// TIA Portal V15.1 export
// export: Created 2024-05-17T05:38:55.5837031Z, ExportSetting WithDefaults, DisplayName Totally Integrated Automation Portal, DisplayVersion V15.1 Update 5, DisplayName TIA Portal Openness, DisplayVersion V15.1 Update 5, DisplayName SINAMICS Startdrive Advanced, DisplayVersion V15.1, DisplayName G130, G150, S120, S150, SINAMICS MV, S210, DisplayVersion V15.1, DisplayName G110M, G120, G120C, G120D, G120P, DisplayVersion V15.1, DisplayName STEP 7 Professional, DisplayVersion V15.1 Update 5, DisplayName STEP 7 Safety, DisplayVersion V15.1, DisplayName WinCC Professional, DisplayVersion V15.1 Update 5, DisplayName SIMATIC Visualization Architect, DisplayVersion V15.1
FUNCTION "209220ZM01DataHandling" : Void   // FC354, FBD
TITLE = 209220ZM01 Data Handling
{ S7_Optimized_Access := 'FALSE' }
AUTHOR : VCC
VERSION : 0.1
// stored: AutoNumber false, IsIECCheckEnabled false, SetENOAutomatically False, UDAEnableTagReadback false
   VAR_OUTPUT
      O_AlarmA : Bool;   // Alarm A
      O_AlarmB : Bool;   // Alarm B
      O_AlarmC : Bool;   // Alarm C
      O_AlarmD : Bool;   // Alarm D
      O_AlarmABCondition : Bool;   // Alarm AB Condition
      H_IAnim : Word;   // Icon Animation
   END_VAR
BEGIN

REGION Network 1: **** 4.6 - Machine status - Indications **** Icon animation
   // Icon animation
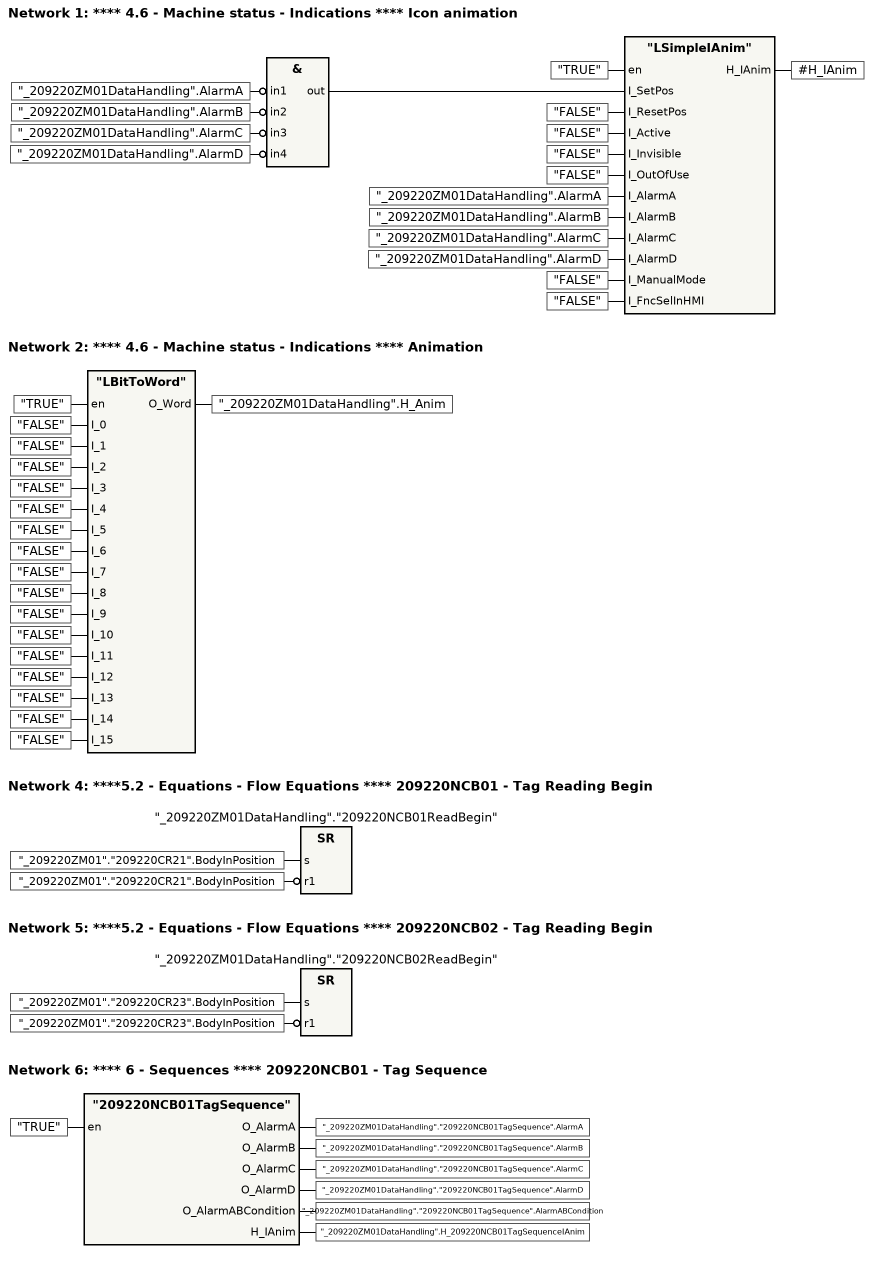
   IF "TRUE" THEN
       "LSimpleIAnim"(I_SetPos := NOT "_209220ZM01DataHandling".AlarmA AND NOT "_209220ZM01DataHandling".AlarmB AND NOT "_209220ZM01DataHandling".AlarmC AND NOT "_209220ZM01DataHandling".AlarmD,
                      I_ResetPos := "FALSE",
                      I_Active := "FALSE",
                      I_Invisible := "FALSE",
                      I_OutOfUse := "FALSE",
                      I_AlarmA := "_209220ZM01DataHandling".AlarmA,
                      I_AlarmB := "_209220ZM01DataHandling".AlarmB,
                      I_AlarmC := "_209220ZM01DataHandling".AlarmC,
                      I_AlarmD := "_209220ZM01DataHandling".AlarmD,
                      I_ManualMode := "FALSE",
                      I_FncSelInHMI := "FALSE",
                      H_IAnim => #H_IAnim);
   END_IF;
END_REGION

REGION Network 2: **** 4.6 - Machine status - Indications **** Animation
   // Animation
   IF "TRUE" THEN
       "LBitToWord"(I_0 := "FALSE",
                    I_1 := "FALSE",
                    I_2 := "FALSE",
                    I_3 := "FALSE",
                    I_4 := "FALSE",
                    I_5 := "FALSE",
                    I_6 := "FALSE",
                    I_7 := "FALSE",
                    I_8 := "FALSE",
                    I_9 := "FALSE",
                    I_10 := "FALSE",
                    I_11 := "FALSE",
                    I_12 := "FALSE",
                    I_13 := "FALSE",
                    I_14 := "FALSE",
                    I_15 := "FALSE",
                    O_Word => "_209220ZM01DataHandling".H_Anim);
   END_IF;
END_REGION

NETWORK
TITLE = **** 4.6 - Machine Status - Indications **** Animation DB number
// DB number
      OPN   "_209220ZM01DataHandling";
      L     DBNO;
      T     "_209220ZM01DataHandling".H_DBnr;

REGION Network 4: ****5.2 - Equations - Flow Equations **** 209220NCB01 - Tag Reading Begin
   // Singal to start the reading of the Tag
   IF "_209220ZM01"."209220CR21".BodyInPosition THEN
       "_209220ZM01DataHandling"."209220NCB01ReadBegin" := TRUE;   // SR flip-flop
   END_IF;
   IF NOT "_209220ZM01"."209220CR21".BodyInPosition THEN
       "_209220ZM01DataHandling"."209220NCB01ReadBegin" := FALSE;
   END_IF;
END_REGION

REGION Network 5: ****5.2 - Equations - Flow Equations **** 209220NCB02 - Tag Reading Begin
   // Singal to start the reading of the Tag
   IF "_209220ZM01"."209220CR23".BodyInPosition THEN
       "_209220ZM01DataHandling"."209220NCB02ReadBegin" := TRUE;   // SR flip-flop
   END_IF;
   IF NOT "_209220ZM01"."209220CR23".BodyInPosition THEN
       "_209220ZM01DataHandling"."209220NCB02ReadBegin" := FALSE;
   END_IF;
END_REGION

REGION Network 6: **** 6 - Sequences **** 209220NCB01 - Tag Sequence
   // Tag Sequence
   IF "TRUE" THEN
       "209220NCB01TagSequence"(O_AlarmA => "_209220ZM01DataHandling"."209220NCB01TagSequence".AlarmA,
                               O_AlarmB => "_209220ZM01DataHandling"."209220NCB01TagSequence".AlarmB,
                               O_AlarmC => "_209220ZM01DataHandling"."209220NCB01TagSequence".AlarmC,
                               O_AlarmD => "_209220ZM01DataHandling"."209220NCB01TagSequence".AlarmD,
                               O_AlarmABCondition => "_209220ZM01DataHandling"."209220NCB01TagSequence".AlarmABCondition,
                               H_IAnim => "_209220ZM01DataHandling".H_209220NCB01TagSequenceIAnim);
   END_IF;
END_REGION

REGION Network 7: **** 6 - Sequences **** 209220NCB02 - Tag Sequence
   // Tag Sequence
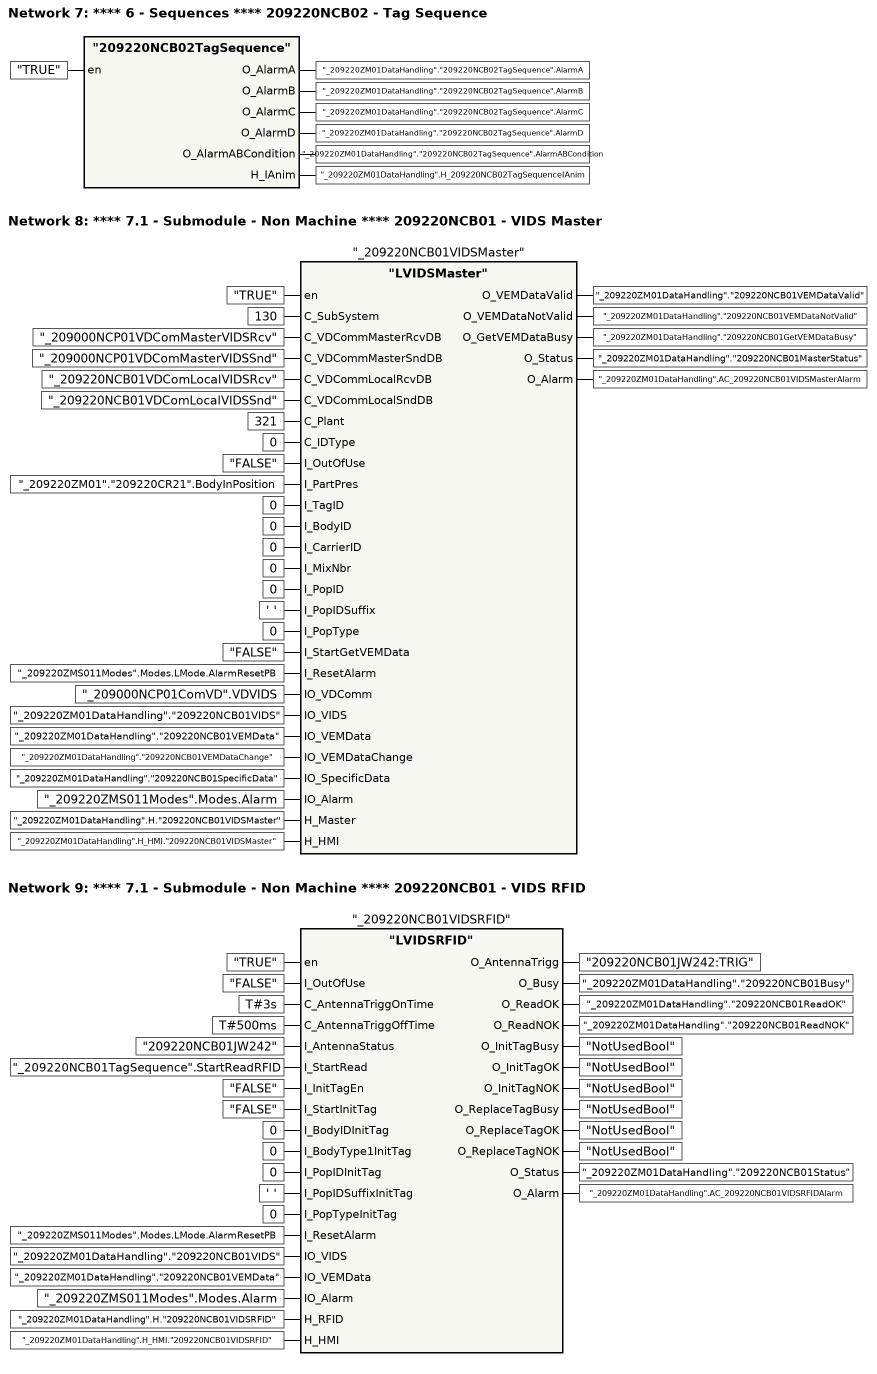
   IF "TRUE" THEN
       "209220NCB02TagSequence"(O_AlarmA => "_209220ZM01DataHandling"."209220NCB02TagSequence".AlarmA,
                               O_AlarmB => "_209220ZM01DataHandling"."209220NCB02TagSequence".AlarmB,
                               O_AlarmC => "_209220ZM01DataHandling"."209220NCB02TagSequence".AlarmC,
                               O_AlarmD => "_209220ZM01DataHandling"."209220NCB02TagSequence".AlarmD,
                               O_AlarmABCondition => "_209220ZM01DataHandling"."209220NCB02TagSequence".AlarmABCondition,
                               H_IAnim => "_209220ZM01DataHandling".H_209220NCB02TagSequenceIAnim);
   END_IF;
END_REGION

REGION Network 8: **** 7.1 - Submodule - Non Machine **** 209220NCB01 - VIDS Master
   // VIDS Master Module
   IF "TRUE" THEN
       "_209220NCB01VIDSMaster"(C_SubSystem := 130,   // "LVIDSMaster"
                               C_VDCommMasterRcvDB := "_209000NCP01VDComMasterVIDSRcv",
                               C_VDCommMasterSndDB := "_209000NCP01VDComMasterVIDSSnd",
                               C_VDCommLocalRcvDB := "_209220NCB01VDComLocalVIDSRcv",
                               C_VDCommLocalSndDB := "_209220NCB01VDComLocalVIDSSnd",
                               C_Plant := 321,
                               C_IDType := 0,
                               I_OutOfUse := "FALSE",
                               I_PartPres := "_209220ZM01"."209220CR21".BodyInPosition,
                               I_TagID := 0,
                               I_BodyID := 0,
                               I_CarrierID := 0,
                               I_MixNbr := 0,
                               I_PopID := 0,
                               I_PopIDSuffix := ' ',
                               I_PopType := 0,
                               I_StartGetVEMData := "FALSE",
                               I_ResetAlarm := "_209220ZMS011Modes".Modes.LMode.AlarmResetPB,
                               IO_VDComm := "_209000NCP01ComVD".VDVIDS,
                               IO_VIDS := "_209220ZM01DataHandling"."209220NCB01VIDS",
                               IO_VEMData := "_209220ZM01DataHandling"."209220NCB01VEMData",
                               IO_VEMDataChange := "_209220ZM01DataHandling"."209220NCB01VEMDataChange",
                               IO_SpecificData := "_209220ZM01DataHandling"."209220NCB01SpecificData",
                               IO_Alarm := "_209220ZMS011Modes".Modes.Alarm,
                               H_Master := "_209220ZM01DataHandling".H."209220NCB01VIDSMaster",
                               H_HMI := "_209220ZM01DataHandling".H_HMI."209220NCB01VIDSMaster",
                               O_VEMDataValid => "_209220ZM01DataHandling"."209220NCB01VEMDataValid",
                               O_VEMDataNotValid => "_209220ZM01DataHandling"."209220NCB01VEMDataNotValid",
                               O_GetVEMDataBusy => "_209220ZM01DataHandling"."209220NCB01GetVEMDataBusy",
                               O_Status => "_209220ZM01DataHandling"."209220NCB01MasterStatus",
                               O_Alarm => "_209220ZM01DataHandling".AC_209220NCB01VIDSMasterAlarm);
   END_IF;
END_REGION

REGION Network 9: **** 7.1 - Submodule - Non Machine **** 209220NCB01 - VIDS RFID
   // VIDS RFID Module
   IF "TRUE" THEN
       "_209220NCB01VIDSRFID"(I_OutOfUse := "FALSE",   // "LVIDSRFID"
                              C_AntennaTriggOnTime := T#3s,
                              C_AntennaTriggOffTime := T#500ms,
                              I_AntennaStatus := "209220NCB01JW242",
                              I_StartRead := "_209220NCB01TagSequence".StartReadRFID,
                              I_InitTagEn := "FALSE",
                              I_StartInitTag := "FALSE",
                              I_BodyIDInitTag := 0,
                              I_BodyType1InitTag := 0,
                              I_PopIDInitTag := 0,
                              I_PopIDSuffixInitTag := ' ',
                              I_PopTypeInitTag := 0,
                              I_ResetAlarm := "_209220ZMS011Modes".Modes.LMode.AlarmResetPB,
                              IO_VIDS := "_209220ZM01DataHandling"."209220NCB01VIDS",
                              IO_VEMData := "_209220ZM01DataHandling"."209220NCB01VEMData",
                              IO_Alarm := "_209220ZMS011Modes".Modes.Alarm,
                              H_RFID := "_209220ZM01DataHandling".H."209220NCB01VIDSRFID",
                              H_HMI := "_209220ZM01DataHandling".H_HMI."209220NCB01VIDSRFID",
                              O_AntennaTrigg => "209220NCB01JW242:TRIG",
                              O_Busy => "_209220ZM01DataHandling"."209220NCB01Busy",
                              O_ReadOK => "_209220ZM01DataHandling"."209220NCB01ReadOK",
                              O_ReadNOK => "_209220ZM01DataHandling"."209220NCB01ReadNOK",
                              O_InitTagBusy => "NotUsedBool",
                              O_InitTagOK => "NotUsedBool",
                              O_InitTagNOK => "NotUsedBool",
                              O_ReplaceTagBusy => "NotUsedBool",
                              O_ReplaceTagOK => "NotUsedBool",
                              O_ReplaceTagNOK => "NotUsedBool",
                              O_Status => "_209220ZM01DataHandling"."209220NCB01Status",
                              O_Alarm => "_209220ZM01DataHandling".AC_209220NCB01VIDSRFIDAlarm);
   END_IF;
END_REGION

REGION Network 10: **** 7.1 - Submodule - Non Machine ****209220NCB01 - VIDS Tracking
   // VIDS Tracking Module
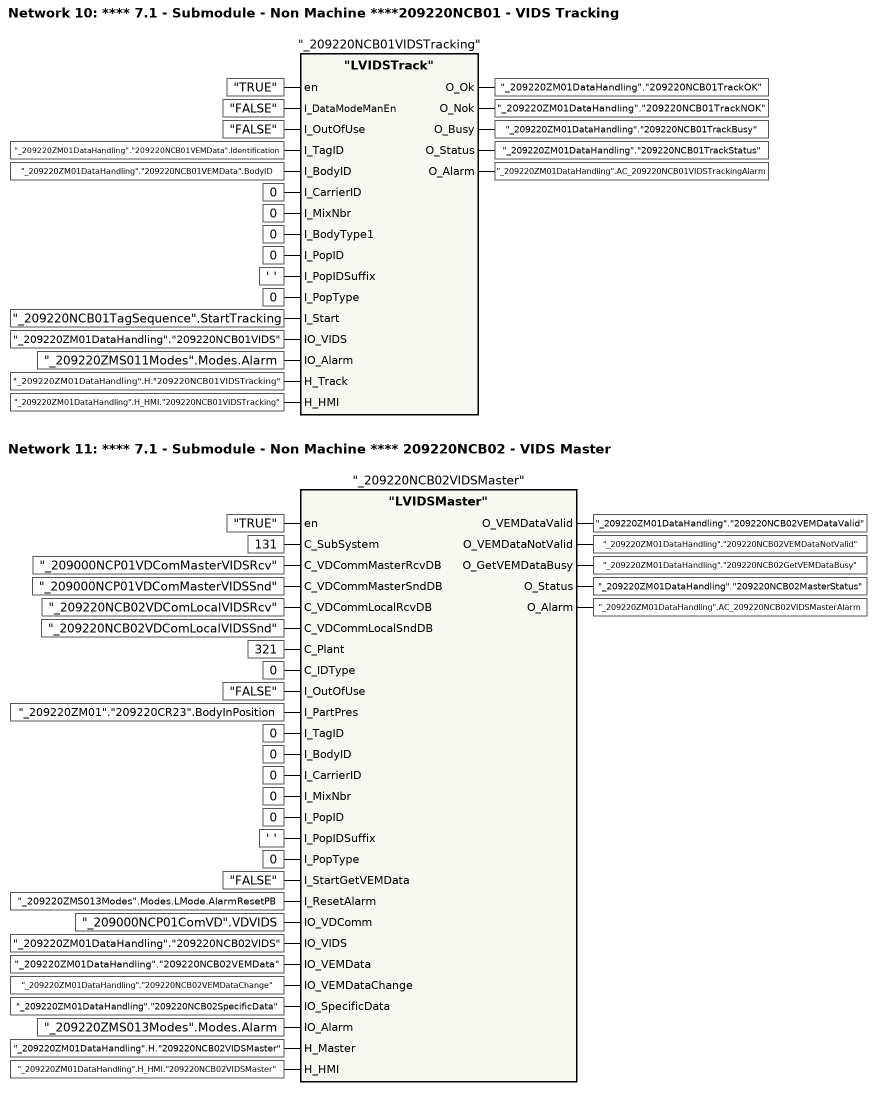
   IF "TRUE" THEN
       "_209220NCB01VIDSTracking"(I_DataModeManEn := "FALSE",   // "LVIDSTrack"
                               I_OutOfUse := "FALSE",
                               I_TagID := "_209220ZM01DataHandling"."209220NCB01VEMData".Identification,
                               I_BodyID := "_209220ZM01DataHandling"."209220NCB01VEMData".BodyID,
                               I_CarrierID := 0,
                               I_MixNbr := 0,
                               I_BodyType1 := 0,
                               I_PopID := 0,
                               I_PopIDSuffix := ' ',
                               I_PopType := 0,
                               I_Start := "_209220NCB01TagSequence".StartTracking,
                               IO_VIDS := "_209220ZM01DataHandling"."209220NCB01VIDS",
                               IO_Alarm := "_209220ZMS011Modes".Modes.Alarm,
                               H_Track := "_209220ZM01DataHandling".H."209220NCB01VIDSTracking",
                               H_HMI := "_209220ZM01DataHandling".H_HMI."209220NCB01VIDSTracking",
                               O_Ok => "_209220ZM01DataHandling"."209220NCB01TrackOK",
                               O_Nok => "_209220ZM01DataHandling"."209220NCB01TrackNOK",
                               O_Busy => "_209220ZM01DataHandling"."209220NCB01TrackBusy",
                               O_Status => "_209220ZM01DataHandling"."209220NCB01TrackStatus",
                               O_Alarm => "_209220ZM01DataHandling".AC_209220NCB01VIDSTrackingAlarm);
   END_IF;
END_REGION

REGION Network 11: **** 7.1 - Submodule - Non Machine **** 209220NCB02 - VIDS Master
   // VIDS Master Module
   IF "TRUE" THEN
       "_209220NCB02VIDSMaster"(C_SubSystem := 131,   // "LVIDSMaster"
                               C_VDCommMasterRcvDB := "_209000NCP01VDComMasterVIDSRcv",
                               C_VDCommMasterSndDB := "_209000NCP01VDComMasterVIDSSnd",
                               C_VDCommLocalRcvDB := "_209220NCB02VDComLocalVIDSRcv",
                               C_VDCommLocalSndDB := "_209220NCB02VDComLocalVIDSSnd",
                               C_Plant := 321,
                               C_IDType := 0,
                               I_OutOfUse := "FALSE",
                               I_PartPres := "_209220ZM01"."209220CR23".BodyInPosition,
                               I_TagID := 0,
                               I_BodyID := 0,
                               I_CarrierID := 0,
                               I_MixNbr := 0,
                               I_PopID := 0,
                               I_PopIDSuffix := ' ',
                               I_PopType := 0,
                               I_StartGetVEMData := "FALSE",
                               I_ResetAlarm := "_209220ZMS013Modes".Modes.LMode.AlarmResetPB,
                               IO_VDComm := "_209000NCP01ComVD".VDVIDS,
                               IO_VIDS := "_209220ZM01DataHandling"."209220NCB02VIDS",
                               IO_VEMData := "_209220ZM01DataHandling"."209220NCB02VEMData",
                               IO_VEMDataChange := "_209220ZM01DataHandling"."209220NCB02VEMDataChange",
                               IO_SpecificData := "_209220ZM01DataHandling"."209220NCB02SpecificData",
                               IO_Alarm := "_209220ZMS013Modes".Modes.Alarm,
                               H_Master := "_209220ZM01DataHandling".H."209220NCB02VIDSMaster",
                               H_HMI := "_209220ZM01DataHandling".H_HMI."209220NCB02VIDSMaster",
                               O_VEMDataValid => "_209220ZM01DataHandling"."209220NCB02VEMDataValid",
                               O_VEMDataNotValid => "_209220ZM01DataHandling"."209220NCB02VEMDataNotValid",
                               O_GetVEMDataBusy => "_209220ZM01DataHandling"."209220NCB02GetVEMDataBusy",
                               O_Status => "_209220ZM01DataHandling"."209220NCB02MasterStatus",
                               O_Alarm => "_209220ZM01DataHandling".AC_209220NCB02VIDSMasterAlarm);
   END_IF;
END_REGION

REGION Network 12: **** 7.1 - Submodule - Non Machine **** 209220NCB02 - VIDS RFID
   // VIDS RFID Module
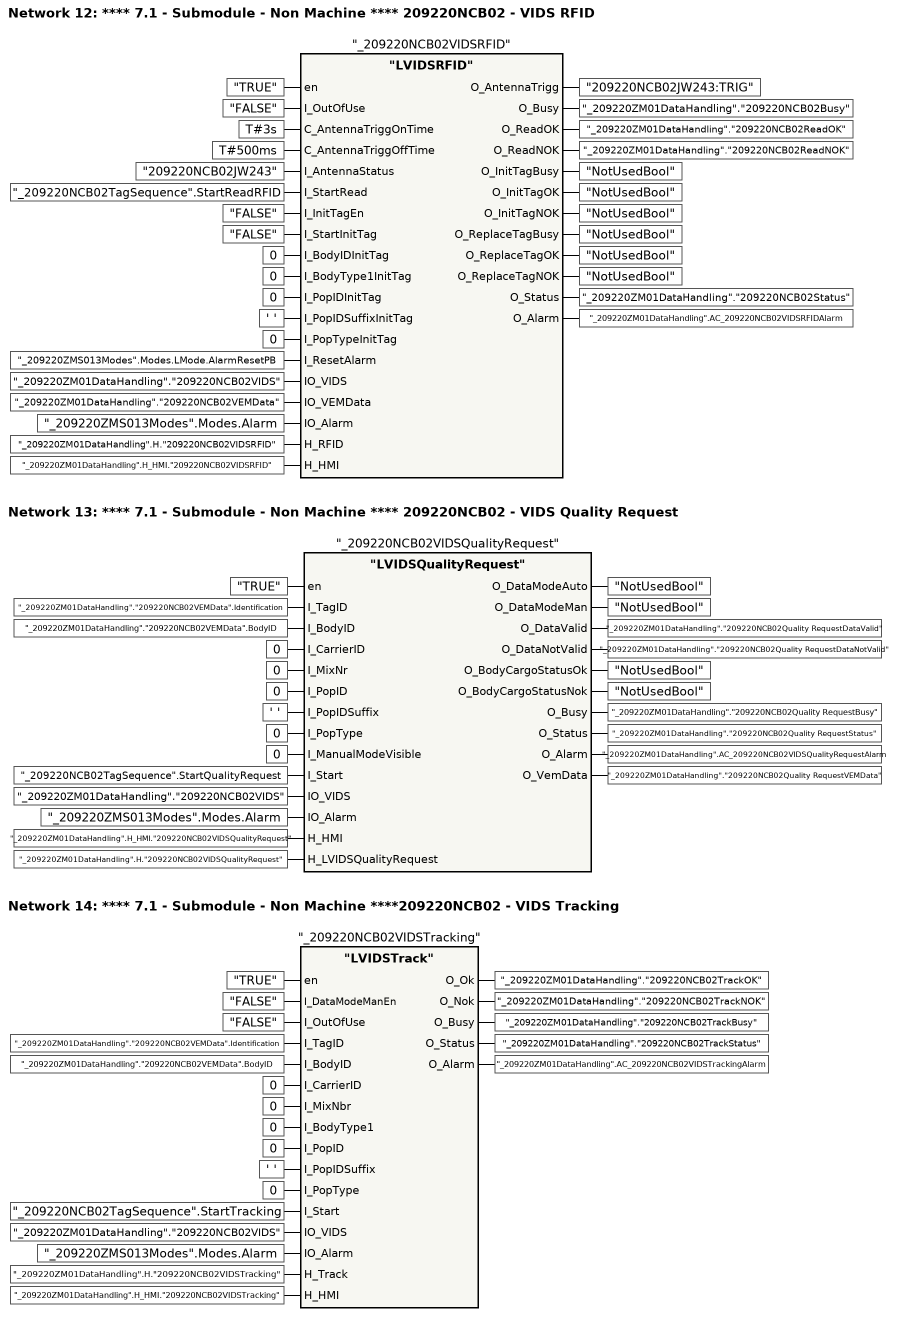
   IF "TRUE" THEN
       "_209220NCB02VIDSRFID"(I_OutOfUse := "FALSE",   // "LVIDSRFID"
                              C_AntennaTriggOnTime := T#3s,
                              C_AntennaTriggOffTime := T#500ms,
                              I_AntennaStatus := "209220NCB02JW243",
                              I_StartRead := "_209220NCB02TagSequence".StartReadRFID,
                              I_InitTagEn := "FALSE",
                              I_StartInitTag := "FALSE",
                              I_BodyIDInitTag := 0,
                              I_BodyType1InitTag := 0,
                              I_PopIDInitTag := 0,
                              I_PopIDSuffixInitTag := ' ',
                              I_PopTypeInitTag := 0,
                              I_ResetAlarm := "_209220ZMS013Modes".Modes.LMode.AlarmResetPB,
                              IO_VIDS := "_209220ZM01DataHandling"."209220NCB02VIDS",
                              IO_VEMData := "_209220ZM01DataHandling"."209220NCB02VEMData",
                              IO_Alarm := "_209220ZMS013Modes".Modes.Alarm,
                              H_RFID := "_209220ZM01DataHandling".H."209220NCB02VIDSRFID",
                              H_HMI := "_209220ZM01DataHandling".H_HMI."209220NCB02VIDSRFID",
                              O_AntennaTrigg => "209220NCB02JW243:TRIG",
                              O_Busy => "_209220ZM01DataHandling"."209220NCB02Busy",
                              O_ReadOK => "_209220ZM01DataHandling"."209220NCB02ReadOK",
                              O_ReadNOK => "_209220ZM01DataHandling"."209220NCB02ReadNOK",
                              O_InitTagBusy => "NotUsedBool",
                              O_InitTagOK => "NotUsedBool",
                              O_InitTagNOK => "NotUsedBool",
                              O_ReplaceTagBusy => "NotUsedBool",
                              O_ReplaceTagOK => "NotUsedBool",
                              O_ReplaceTagNOK => "NotUsedBool",
                              O_Status => "_209220ZM01DataHandling"."209220NCB02Status",
                              O_Alarm => "_209220ZM01DataHandling".AC_209220NCB02VIDSRFIDAlarm);
   END_IF;
END_REGION

REGION Network 13: **** 7.1 - Submodule - Non Machine **** 209220NCB02 - VIDS Quality Request
   IF "TRUE" THEN
       "_209220NCB02VIDSQualityRequest"(I_TagID := "_209220ZM01DataHandling"."209220NCB02VEMData".Identification,   // "LVIDSQualityRequest"
                               I_BodyID := "_209220ZM01DataHandling"."209220NCB02VEMData".BodyID,
                               I_CarrierID := 0,
                               I_MixNr := 0,
                               I_PopID := 0,
                               I_PopIDSuffix := ' ',
                               I_PopType := 0,
                               I_ManualModeVisible := 0,
                               I_Start := "_209220NCB02TagSequence".StartQualityRequest,
                               IO_VIDS := "_209220ZM01DataHandling"."209220NCB02VIDS",
                               IO_Alarm := "_209220ZMS013Modes".Modes.Alarm,
                               H_HMI := "_209220ZM01DataHandling".H_HMI."209220NCB02VIDSQualityRequest",
                               H_LVIDSQualityRequest := "_209220ZM01DataHandling".H."209220NCB02VIDSQualityRequest",
                               O_DataModeAuto => "NotUsedBool",
                               O_DataModeMan => "NotUsedBool",
                               O_DataValid => "_209220ZM01DataHandling"."209220NCB02Quality RequestDataValid",
                               O_DataNotValid => "_209220ZM01DataHandling"."209220NCB02Quality RequestDataNotValid",
                               O_BodyCargoStatusOk => "NotUsedBool",
                               O_BodyCargoStatusNok => "NotUsedBool",
                               O_Busy => "_209220ZM01DataHandling"."209220NCB02Quality RequestBusy",
                               O_Status => "_209220ZM01DataHandling"."209220NCB02Quality RequestStatus",
                               O_Alarm => "_209220ZM01DataHandling".AC_209220NCB02VIDSQualityRequestAlarm,
                               O_VemData => "_209220ZM01DataHandling"."209220NCB02Quality RequestVEMData");
   END_IF;
END_REGION

REGION Network 14: **** 7.1 - Submodule - Non Machine ****209220NCB02 - VIDS Tracking
   // VIDS Tracking Module
   IF "TRUE" THEN
       "_209220NCB02VIDSTracking"(I_DataModeManEn := "FALSE",   // "LVIDSTrack"
                               I_OutOfUse := "FALSE",
                               I_TagID := "_209220ZM01DataHandling"."209220NCB02VEMData".Identification,
                               I_BodyID := "_209220ZM01DataHandling"."209220NCB02VEMData".BodyID,
                               I_CarrierID := 0,
                               I_MixNbr := 0,
                               I_BodyType1 := 0,
                               I_PopID := 0,
                               I_PopIDSuffix := ' ',
                               I_PopType := 0,
                               I_Start := "_209220NCB02TagSequence".StartTracking,
                               IO_VIDS := "_209220ZM01DataHandling"."209220NCB02VIDS",
                               IO_Alarm := "_209220ZMS013Modes".Modes.Alarm,
                               H_Track := "_209220ZM01DataHandling".H."209220NCB02VIDSTracking",
                               H_HMI := "_209220ZM01DataHandling".H_HMI."209220NCB02VIDSTracking",
                               O_Ok => "_209220ZM01DataHandling"."209220NCB02TrackOK",
                               O_Nok => "_209220ZM01DataHandling"."209220NCB02TrackNOK",
                               O_Busy => "_209220ZM01DataHandling"."209220NCB02TrackBusy",
                               O_Status => "_209220ZM01DataHandling"."209220NCB02TrackStatus",
                               O_Alarm => "_209220ZM01DataHandling".AC_209220NCB02VIDSTrackingAlarm);
   END_IF;
END_REGION

REGION Network 15: **** 9 - Alarm Summary **** Alarm AB Condition
   // Alarm AB Condition
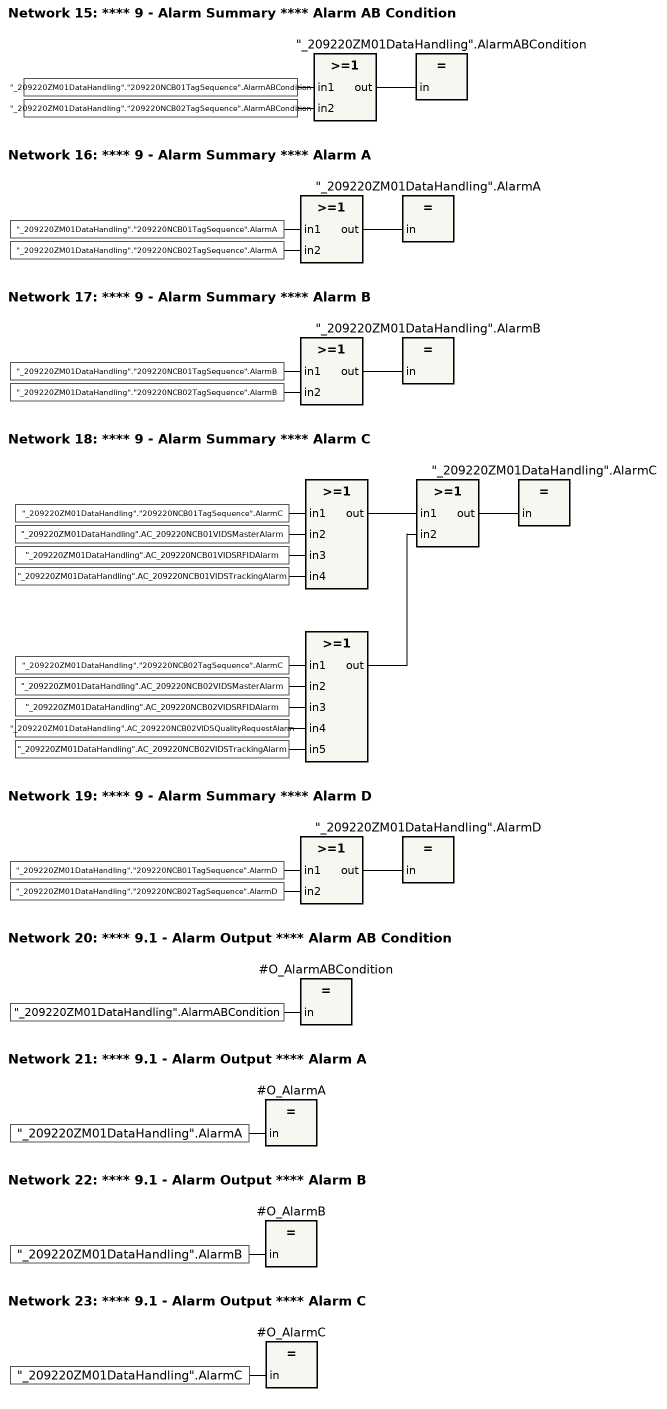
   "_209220ZM01DataHandling".AlarmABCondition := "_209220ZM01DataHandling"."209220NCB01TagSequence".AlarmABCondition OR "_209220ZM01DataHandling"."209220NCB02TagSequence".AlarmABCondition;
END_REGION

REGION Network 16: **** 9 - Alarm Summary **** Alarm A
   // Alarm A
   "_209220ZM01DataHandling".AlarmA := "_209220ZM01DataHandling"."209220NCB01TagSequence".AlarmA OR "_209220ZM01DataHandling"."209220NCB02TagSequence".AlarmA;
END_REGION

REGION Network 17: **** 9 - Alarm Summary **** Alarm B
   // Alarm B
   "_209220ZM01DataHandling".AlarmB := "_209220ZM01DataHandling"."209220NCB01TagSequence".AlarmB OR "_209220ZM01DataHandling"."209220NCB02TagSequence".AlarmB;
END_REGION

REGION Network 18: **** 9 - Alarm Summary **** Alarm C
   // Alarm C
   "_209220ZM01DataHandling".AlarmC := "_209220ZM01DataHandling"."209220NCB01TagSequence".AlarmC OR "_209220ZM01DataHandling".AC_209220NCB01VIDSMasterAlarm OR "_209220ZM01DataHandling".AC_209220NCB01VIDSRFIDAlarm OR "_209220ZM01DataHandling".AC_209220NCB01VIDSTrackingAlarm OR "_209220ZM01DataHandling"."209220NCB02TagSequence".AlarmC OR "_209220ZM01DataHandling".AC_209220NCB02VIDSMasterAlarm OR "_209220ZM01DataHandling".AC_209220NCB02VIDSRFIDAlarm OR "_209220ZM01DataHandling".AC_209220NCB02VIDSQualityRequestAlarm OR "_209220ZM01DataHandling".AC_209220NCB02VIDSTrackingAlarm;
END_REGION

REGION Network 19: **** 9 - Alarm Summary **** Alarm D
   // Alarm D
   "_209220ZM01DataHandling".AlarmD := "_209220ZM01DataHandling"."209220NCB01TagSequence".AlarmD OR "_209220ZM01DataHandling"."209220NCB02TagSequence".AlarmD;
END_REGION

REGION Network 20: **** 9.1 - Alarm Output **** Alarm AB Condition
   // Alarm AB Condition
   #O_AlarmABCondition := "_209220ZM01DataHandling".AlarmABCondition;
END_REGION

REGION Network 21: **** 9.1 - Alarm Output **** Alarm A
   // Alarm A
   #O_AlarmA := "_209220ZM01DataHandling".AlarmA;
END_REGION

REGION Network 22: **** 9.1 - Alarm Output **** Alarm B
   // Alarm B
   #O_AlarmB := "_209220ZM01DataHandling".AlarmB;
END_REGION

REGION Network 23: **** 9.1 - Alarm Output **** Alarm C
   // Alarm C
   #O_AlarmC := "_209220ZM01DataHandling".AlarmC;
END_REGION

REGION Network 24: **** 9.1 - Alarm Output **** Alarm D
   // Alarm D
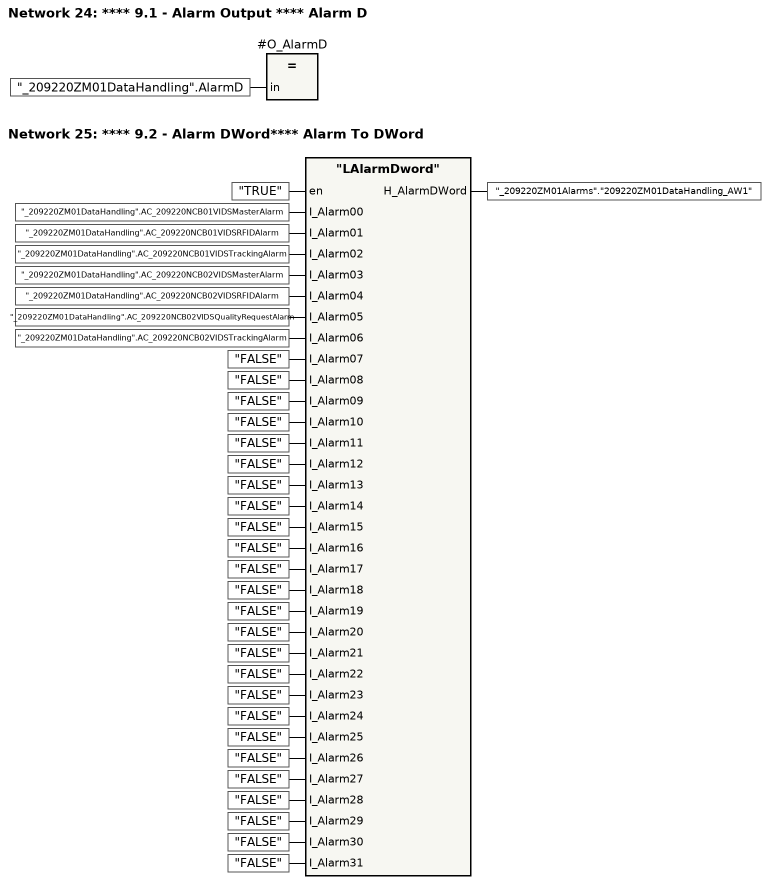
   #O_AlarmD := "_209220ZM01DataHandling".AlarmD;
END_REGION

REGION Network 25: **** 9.2 - Alarm DWord**** Alarm To DWord
   // Alarm Word
   IF "TRUE" THEN
       "LAlarmDword"(I_Alarm00 := "_209220ZM01DataHandling".AC_209220NCB01VIDSMasterAlarm,
                     I_Alarm01 := "_209220ZM01DataHandling".AC_209220NCB01VIDSRFIDAlarm,
                     I_Alarm02 := "_209220ZM01DataHandling".AC_209220NCB01VIDSTrackingAlarm,
                     I_Alarm03 := "_209220ZM01DataHandling".AC_209220NCB02VIDSMasterAlarm,
                     I_Alarm04 := "_209220ZM01DataHandling".AC_209220NCB02VIDSRFIDAlarm,
                     I_Alarm05 := "_209220ZM01DataHandling".AC_209220NCB02VIDSQualityRequestAlarm,
                     I_Alarm06 := "_209220ZM01DataHandling".AC_209220NCB02VIDSTrackingAlarm,
                     I_Alarm07 := "FALSE",
                     I_Alarm08 := "FALSE",
                     I_Alarm09 := "FALSE",
                     I_Alarm10 := "FALSE",
                     I_Alarm11 := "FALSE",
                     I_Alarm12 := "FALSE",
                     I_Alarm13 := "FALSE",
                     I_Alarm14 := "FALSE",
                     I_Alarm15 := "FALSE",
                     I_Alarm16 := "FALSE",
                     I_Alarm17 := "FALSE",
                     I_Alarm18 := "FALSE",
                     I_Alarm19 := "FALSE",
                     I_Alarm20 := "FALSE",
                     I_Alarm21 := "FALSE",
                     I_Alarm22 := "FALSE",
                     I_Alarm23 := "FALSE",
                     I_Alarm24 := "FALSE",
                     I_Alarm25 := "FALSE",
                     I_Alarm26 := "FALSE",
                     I_Alarm27 := "FALSE",
                     I_Alarm28 := "FALSE",
                     I_Alarm29 := "FALSE",
                     I_Alarm30 := "FALSE",
                     I_Alarm31 := "FALSE",
                     H_AlarmDWord => "_209220ZM01Alarms"."209220ZM01DataHandling_AW1");
   END_IF;
END_REGION
END_FUNCTION
